// TIA Portal V20 export
TYPE "LER_typeStatusOutputCam"
// stored: Access Published
   STRUCT
      CamOutput : Bool;
      Busy : Bool;
      Error : Bool;
      ErrorId : Word;
   END_STRUCT;
END_TYPE
